FUNCTION_BLOCK E_CTD (* Event-Driven Down Counter *)
  (* Standard: 61499-1-A.1; Classification: Event-driven blocks; Function: Down-counter *)
  (* Version 0.0, 2006-09-07, JHC, Holobloc Inc *)
  (* Compiler header: package fb.rt.events; *)
  (* Compiler Java Sun JDK 1.5.0 *)
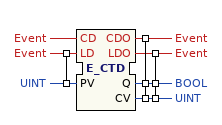
  EVENT_INPUT
    CD; (* Count Down *)
    LD WITH PV; (* Load PV to CV *)
  END_EVENT
  EVENT_OUTPUT
    CDO WITH Q, CV; (* Count Down Output Event *)
    LDO WITH Q, CV; (* Load Output Event *)
  END_EVENT
  VAR_INPUT
    PV : UINT; (* Preset Value *)
  END_VAR
  VAR_OUTPUT
    Q : BOOL; (* CV==0 *)
    CV : UINT;
  END_VAR
END_FUNCTION_BLOCK
